(* IEC 61131-3 sources: Learning-PLC/Openplc/pous/programs, 1 file *)

(* ---- main.st ---- *)
PROGRAM main
  VAR
  END_VAR

for i := 0 to 10 do

end_for;

END_PROGRAM
